SUBAPPLICATION Uebung_246_AX (* logiBUS_IXA I1(Hoch)/I2(Runter) auf 3-Stufen-Sollwert 75%/25%/50%(Neutral), zwei AR_AX_SEL_AR verkettet *)
  (* Standard: 61499-2; Description: Copyright (c) 2026 Meisterschulen am Ostbahnhof This program and the accompanying materials are made available under the terms of the Eclipse Public License 2.0 which is available at https://www.eclipse.org/legal/epl-2.0/ SPDX-License-Identifier: EPL-2.0 *)
  (* Version 1.0, 2026-09-07, Franz Höpfinger, Meisterschulen am Ostbahnhof, initial API and implementation and/or initial documentation *)
  PACKAGE Uebungen;
  IMPORT logiBUS::io::DI::logiBUS_DI::Input_I1;
  IMPORT logiBUS::io::DI::logiBUS_DI::Input_I2;
  IMPORT Uebungen::const::UT::DefaultPool_Numeric::OutputNumber_N3_N;
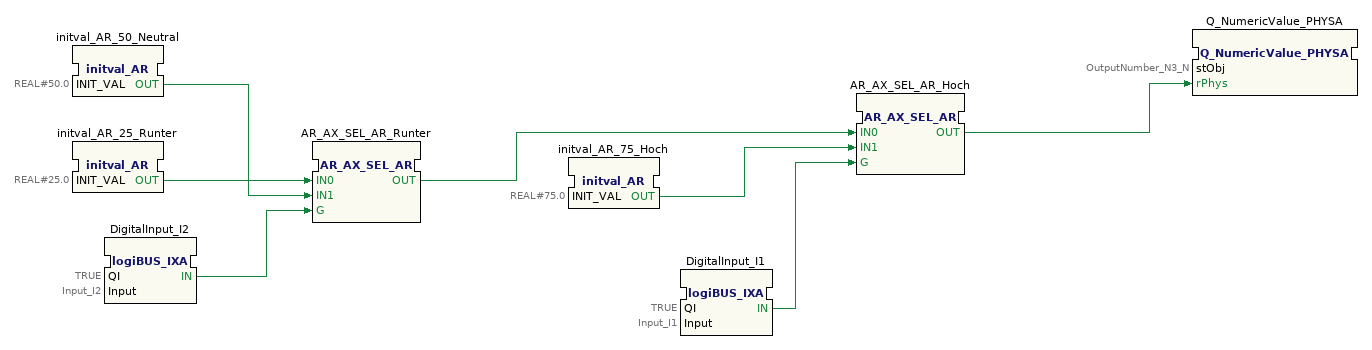
  (* Zwei verkettete Binaer-Selektoren statt eines 3-Wege-Selektors (den es fuer AR nicht gibt): innen waehlt I2 (Runter) zwischen Neutral(50) und Runter(25), aussen waehlt I1 (Hoch) zwischen diesem Ergebnis und Hoch(75). Werden I1 und I2 gleichzeitig gehalten, gewinnt I1 (Hoch), weil sein Selektor der aeussere ist - bewusste Prioritaet, siehe Beschreibung. *)
  FBS
    DigitalInput_I1 : logiBUS::io::DI::logiBUS_IXA(QI := TRUE, Input := Input_I1);
    DigitalInput_I2 : logiBUS::io::DI::logiBUS_IXA(QI := TRUE, Input := Input_I2);
    initval_AR_50_Neutral : adapter::types::unidirectional::AR::initval::initval_AR(INIT_VAL := REAL#50.0);
    initval_AR_25_Runter : adapter::types::unidirectional::AR::initval::initval_AR(INIT_VAL := REAL#25.0);
    initval_AR_75_Hoch : adapter::types::unidirectional::AR::initval::initval_AR(INIT_VAL := REAL#75.0);
    AR_AX_SEL_AR_Runter : adapter::iec61131::selection::AR_AX_SEL_AR;
    AR_AX_SEL_AR_Hoch : adapter::iec61131::selection::AR_AX_SEL_AR;
    Q_NumericValue_PHYSA : isobus::UT::Q::Q_NumericValue_PHYSA(stObj := OutputNumber_N3_N);
  END_FBS
  ADAPTER_CONNECTIONS
    initval_AR_50_Neutral.OUT TO AR_AX_SEL_AR_Runter.IN0;
    initval_AR_25_Runter.OUT TO AR_AX_SEL_AR_Runter.IN1;
    DigitalInput_I2.IN TO AR_AX_SEL_AR_Runter.G;
    AR_AX_SEL_AR_Runter.OUT TO AR_AX_SEL_AR_Hoch.IN0;
    initval_AR_75_Hoch.OUT TO AR_AX_SEL_AR_Hoch.IN1;
    DigitalInput_I1.IN TO AR_AX_SEL_AR_Hoch.G;
    AR_AX_SEL_AR_Hoch.OUT TO Q_NumericValue_PHYSA.rPhys;
  END_CONNECTIONS
END_SUBAPPLICATION
